(* IEC 61131-3 sources: HappyLearnCodesys/content/softmotion/Robotics_DynamicModel, 17 files *)

(* ---- MatSI_ApplyTwist.st ---- *)
/// Applies a spatial inertia matrix to a twist vector
/// resulting in a generalized momentum or force vector
/// depending on whether the twist represents a velocity
/// or an acceleration.
FUNCTION MatSI_ApplyTwist
VAR_IN_OUT
    /// The resulting generalized momentum or force.
    W : WrenchVec;
END_VAR
VAR_IN_OUT CONSTANT
    /// The spatial inertia matrix.
    G : SMDYN.DynSpatialInertia;
    /// The generalized velocity or acceleration.
    T : TwistVec;
END_VAR

SM3M.SMC_Matrix3_Apply(W.m, G.I, T.w);
SM3M.SMC_V3_Mult(W.f, T.v, G.m);

(* ---- SMC_Frame_ApplyTwist.st ---- *)
/// Applies a coordinate transformation T_ab to a twist vector V_b in se(3).
///       |   mR     0 |
/// V_a = |            | V_b
///       |[vT]*mR   mR|
FUNCTION SMC_Frame_ApplyTwist
VAR_IN_OUT
    /// Twist vector in a frame coordinates
	V_a : TwistVec;
END_VAR
VAR_IN_OUT CONSTANT
    /// Orientation and position of the b frame
    /// in a frame coordinates.
	T_ab : SM3M.SMC_Frame;
    /// Twist vector in b frame coordinates.
	V_b : TwistVec;
END_VAR
VAR
    vTmp : SM3M.SMC_VECTOR3D;
END_VAR

SM3M.SMC_Matrix3_Apply(V_a.w, T_ab.mR, V_b.w);
SM3M.SMC_Matrix3_Apply(V_a.v, T_ab.mR, V_b.v);
SM3M.SMC_V3_Cross(vTmp, T_ab.vT, V_a.w);
SM3M.SMC_V3_Add(V_a.v, V_a.v, vTmp);

(* ---- SMC_Frame_ApplyWrench.st ---- *)
/// Applies a coordinate transformation T_ab to a wrench vector F_a in se(3).
///       |mR^T  mR^T*[vT]^T|
/// F_b = |                 | F_a
///       | 0         mR^T  |
FUNCTION SMC_Frame_ApplyWrench
VAR_IN_OUT
    /// Wrench vector in b frame coordinates.
	F_b : WrenchVec;
END_VAR
VAR_IN_OUT CONSTANT
    /// Orientation and position of the b frame
    /// in a frame coordinates.
	T_ab : SM3M.SMC_Frame;
    /// Wrench vector in a frame coordinates.
	F_a : WrenchVec;
END_VAR
VAR
    mR_ : SM3M.SMC_Matrix3;
    wTmp0 : SM3M.SMC_VECTOR3D;
    wTmp1 : SM3M.SMC_VECTOR3D;
END_VAR

SM3M.SMC_Matrix3_Transpose(mR_, T_ab.mR);
SM3M.SMC_Matrix3_Apply(F_b.m, mR_, F_a.m);
SM3M.SMC_V3_Cross(wTmp0, T_ab.vT, F_a.f);
SM3M.SMC_Matrix3_Apply(wTmp1, mR_, wTmp0);
SM3M.SMC_V3_Sub(F_b.m, F_b.m, wTmp1);

SM3M.SMC_Matrix3_Apply(F_b.f, mR_, F_a.f);

(* ---- SMC_Frame_FromScrewAxisAngle.st ---- *)
/// Calculates an SE(3) frame from a screw axis
/// (a normalized |TwistVec|) and an angle.
FUNCTION SMC_Frame_FromScrewAxisAngle
VAR_IN_OUT
    /// The resulting frame.
    f : SM3M.SMC_Frame;
END_VAR
VAR_IN_OUT CONSTANT
    /// The screw axis.
    A : TwistVec;
END_VAR
VAR_INPUT
    /// The angle.
    theta : LREAL;
END_VAR
VAR
    wv : SM3M.SMC_VECTOR3D;
    w2v : SM3M.SMC_VECTOR3D;
    wt : SM3M.SMC_VECTOR3D;
END_VAR

SM3M.SMC_V3_Cross(wv, A.w, A.v);
SM3M.SMC_V3_Cross(w2v, A.w, wv);

SM3M.SMC_V3_Mult(f.vT, A.v, theta);
SM3M.SMC_V3_MAdd(f.vT, f.vT, wv, (1 - COS(theta)));
SM3M.SMC_V3_MAdd(f.vT, f.vT, w2v, (theta - SIN(theta)));

SM3M.SMC_V3_Mult(wt, A.w, theta);
SM3M.SMC_Matrix3_FromAxisAngle(f.mR, wt);

(* ---- SMC_OpenChainKinematics_SolveForward.st ---- *)
FUNCTION SMC_OpenChainKinematics_SolveForward
VAR_IN_OUT
    fTCP : SM3M.SMC_Frame;
END_VAR
VAR_IN_OUT CONSTANT
    aS : ARRAY[0..SM3M.SMC_MAX_VEC_DIM-1] OF TwistVec;
    vJoints : SM3M.SMC_Vec;
    fTCP_init : SM3M.SMC_Frame;
END_VAR
VAR
    i : UDINT;
    fTmp : SM3M.SMC_Frame;
    afCur : ARRAY[0..1] OF SM3M.SMC_Frame;
END_VAR

i := TO_UDINT(vJoints.n);
afCur[i AND 1] := fTCP_init;
WHILE i > 0 DO
    SMC_Frame_FromScrewAxisAngle(fTmp, aS[i-1], vJoints.a[i-1]);
    SM3M.SMC_Frame_Mult(afCur[(i-1) AND 1], fTmp, afCur[i AND 1]);

    i := i - 1;
END_WHILE

fTCP := afCur[0];

(* ---- Twist_Bracket_Twist.st ---- *)
/// Calculates the generalized cross product
/// between two |TwistVec|s, both representing
/// generalized velocities. The result is a
/// generalized acceleration.
FUNCTION Twist_Bracket_Twist
VAR_IN_OUT
    /// The resulting acceleration.
    V_dst : TwistVec;
END_VAR
VAR_IN_OUT CONSTANT
    /// The first velocity.
    V_lhs : TwistVec;
    /// The second velocity.
    V_rhs : TwistVec;
END_VAR
VAR
    v0 : SM3M.SMC_VECTOR3D;
    v1 : SM3M.SMC_VECTOR3D;
END_VAR

SM3M.SMC_V3_Cross(v0, V_lhs.v, V_rhs.w);
SM3M.SMC_V3_Cross(v1, V_lhs.w, V_rhs.v);
SM3M.SMC_V3_Cross(V_dst.w, V_lhs.w, V_rhs.w);
SM3M.SMC_V3_Add(V_dst.v, v0, v1);

(* ---- Twist_Bracket_Wrench.st ---- *)
/// Calculates the generalized cross product
/// between a |TwistVec|, representing a generalized
/// velocity, and a |WrenchVec|, representing a
/// generalized momentum, resulting in a generalized
/// force.
FUNCTION Twist_Bracket_Wrench
VAR_IN_OUT
    /// The resulting force.
    F_dst : WrenchVec;
END_VAR
VAR_IN_OUT CONSTANT
    /// The velocity.
    V_src : TwistVec;
    /// The momentum.
    F_src : WrenchVec;
END_VAR
VAR
    m0 : SM3M.SMC_VECTOR3D;
    m1 : SM3M.SMC_VECTOR3D;
END_VAR

SM3M.SMC_V3_Cross(m0, F_src.m, V_src.w);
SM3M.SMC_V3_Cross(m1, F_src.f, V_src.v);
SM3M.SMC_V3_Cross(F_dst.f, F_src.f, V_src.w);
SM3M.SMC_V3_Add(F_dst.m, m0, m1);

(* ---- TwistVec_Add.st ---- *)
FUNCTION TwistVec_Add
VAR_IN_OUT
    V_dst : TwistVec;
END_VAR
VAR_IN_OUT CONSTANT
    V_lhs : TwistVec;
    V_rhs : TwistVec;
END_VAR

SM3M.SMC_V3_Add(V_dst.w, V_lhs.w, V_rhs.w);
SM3M.SMC_V3_Add(V_dst.v, V_lhs.v, V_rhs.v);

(* ---- TwistVec_Scale.st ---- *)
FUNCTION TwistVec_Scale
VAR_IN_OUT
    V_dst : TwistVec;
END_VAR
VAR_IN_OUT CONSTANT
    V_src : TwistVec;
END_VAR
VAR_INPUT
    theta : LREAL;
END_VAR

SM3M.SMC_V3_Mult(V_dst.w, V_src.w, theta);
SM3M.SMC_V3_Mult(V_dst.v, V_src.v, theta);

(* ---- Wrench_Dot_Twist.st ---- *)
/// Calculates the dot product between a wrench and a twist.
FUNCTION Wrench_Dot_Twist
VAR_IN_OUT CONSTANT
    F : WrenchVec;
    V : TwistVec;
END_VAR
VAR_OUTPUT
    Wrench_Dot_Twist : LREAL;
END_VAR

Wrench_Dot_Twist := SM3M.SMC_V3_Dot(F.m, V.w) + SM3M.SMC_V3_Dot(F.f, V.v);

(* ---- WrenchVec_Add.st ---- *)
FUNCTION WrenchVec_Add
VAR_IN_OUT
    F_dst : WrenchVec;
END_VAR
VAR_IN_OUT CONSTANT
    F_lhs : WrenchVec;
    F_rhs : WrenchVec;
END_VAR

SM3M.SMC_V3_Add(F_dst.m, F_lhs.m, F_rhs.m);
SM3M.SMC_V3_Add(F_dst.f, F_lhs.f, F_rhs.f);

(* ---- WrenchVec_Sub.st ---- *)
FUNCTION WrenchVec_Sub
VAR_IN_OUT
    V_dst : WrenchVec;
END_VAR
VAR_IN_OUT CONSTANT
    V_lhs : WrenchVec;
    V_rhs : WrenchVec;
END_VAR

SM3M.SMC_V3_Sub(V_dst.m, V_lhs.m, V_rhs.m);
SM3M.SMC_V3_Sub(V_dst.f, V_lhs.f, V_rhs.f);

(* ---- DynModel_Scara2_Z.st ---- *)
(*
    檔案用途：
      定義一具 3 自由度 Scara+Z 機構的動力學模型，包含各連桿的幾何尺寸、
      質量、慣性矩與螺旋軸（screw axes），並實作 SMDYN.ISMDynamics 介面，
      供 SoftMotion 的動力學模組計算關節扭矩與負載效應。
    教學重點：
      - 觀察 m_aM（各連桿質心座標）、m_aG（空間慣性）、m_aS（螺旋軸）三組資料的物理意義。
      - 理解 DOF 與臂長／質量等常數，如何對應到實際 Scara 幾何結構。
      - 作為自訂機構動力學定義的範例，供其他機構參考套用。
*)
FUNCTION_BLOCK DynModel_Scara2_Z IMPLEMENTS SMDYN.ISMDynamics
VAR CONSTANT
	/// Degrees of freedom.
	DOF : DINT := 3;
	/// All length values in [m]
	armOneLength : LREAL := 0.4;
	armTwoLength : LREAL := 0.3;
	baseHeight : LREAL := 0.6;
	armOneHeight : LREAL := 0.06;
	armTwoHeight : LREAL := 0.06;
	zAxisLength : LREAL := 0.3;
	zAxisOffset : LREAL := -0.05;
	/// All mass values in [kg]
	armOneMass : LREAL := 3;
	armTwoMass : LREAL := 4;
	zAxisMass : LREAL := 1;

	/// The home position of all link frames. |aM[i]| contains
    /// the frame of the ith link expressed in the coordinates of the
    /// (i-1)th link frame.
    /// All frames are expected to be situated at the link's center
    /// of mass.
    m_aM : ARRAY[0..SMRB.MAX_VEC_DIM] OF SM3M.SMC_Frame := [
        /// All values of vT in [m]
        ///
        /// The center of mass of arm 1 expressed in the base coordinate system 0:
        (mR:= (
            aElems:= [
                1, 0, 0,
                0, -1, 0,
                0, 0, -1]),
         vT:= (dX:= armOneLength / 2.0, dY:= 0, dZ:= baseHeight + armOneHeight / 2.0)),
        /// The center of mass of arm 2 expressed in the coordinate system of arm 1:
        (mR:= (
            aElems:= [
                1, 0, 0,
                0, 1, 0,
                0, 0, 1]),
         vT:= (dX:= armOneLength / 2.0 + armTwoLength / 2.0, dY:= 0, dZ:= armOneHeight / 2.0 + armTwoHeight / 2.0)),
        /// The center of mass of the z-axis expressed in the coordinate system of arm 2:
        (mR:= (
            aElems:= [
                1, 0, 0,
                0, 1, 0,
                0, 0, 1]),
         vT:= (dX:= armTwoLength / 2.0, dY:= 0, dZ:= zAxisLength / 2.0 - armTwoHeight / 2.0 + zAxisOffset)),
        /// One additional array entry, to handle an arbitrary load at the TCP, expressed
		/// in the coordinate system of the z-axis.
        (mR:= (
            aElems:= [
                1, 0, 0,
                0, 1, 0,
                0, 0, 1]),
         vT:= (dX:= 0, dY:= 0, dZ:= - zAxisLength / 2.0))];

	/// The spatial inertia matrices of all links, expressed in the
    /// respectives link's frame.
    m_aG : ARRAY[0..SMRB.MAX_VEC_DIM-1] OF SMDYN.DynSpatialInertia := [
        /// All inertia values in [kg m²]
        /// and all mass values in [kg]
        /// Arm 1
        (I:= (
            aElems:= [
                0, 0, 0,
                0, 1/12.0 * armOneMass * armOneLength * armOneLength, 0,
                0, 0, 1/12.0 * armOneMass * armOneLength * armOneLength]),
         m:= armOneMass),
        /// Arm 2
        (I:= (
            aElems:= [
                0, 0, 0,
                0, 1/12.0 * armTwoMass * armTwoLength * armTwoLength, 0,
                0, 0, 1/12.0 * armTwoMass * armTwoLength * armTwoLength]),
         m:= armTwoMass),
        /// z-axis
        (I:= (
            aElems:= [
                1/12.0 * zAxisMass * zAxisLength * zAxisLength, 0, 0,
                0, 1/12.0 * zAxisMass * zAxisLength * zAxisLength, 0,
                0, 0, 0]),
         m:= zAxisMass)];

	/// The screw axes of all joints, expressed in the base frame.
    m_aS : ARRAY[0..SMRB.MAX_VEC_DIM-1] OF TwistVec := [
		/// Angular velocities in [rad/s] and linear velocities in [m/s].
        /// Screw axis of arm 1
        (w:= (dX:= 0, dY:= 0, dZ:= 1),
         v:= (dX:= 0, dY:= 0, dZ:= 0)),
        /// Screw axis of arm 2
        (w:= (dX:= 0, dY:= 0, dZ:= 1),
         v:= (dX:= 0, dY:= -armOneLength, dZ:= 0)),
        /// Screw axis of the z-axis
        (w:= (dX:= 0, dY:= 0, dZ:= 0),
         v:= (dX:= 0, dY:= 0, dZ:= 1))];
END_VAR
VAR
    /// The home position of all link frames. |m_aM_inv[i]| contains
    /// the frame of the (i-1) link expressed in the coordinates of the
    /// ith link frame.
    /// All frames are expected to be situated at the link's center
    /// of mass.
    m_aM_inv : ARRAY[0..SM3M.SMC_MAX_VEC_DIM] OF SM3M.SMC_Frame;
    /// The screw axes of all joints, expressed in the link's frame.
    m_aA : ARRAY[0..SM3M.SMC_MAX_VEC_DIM-1] OF TwistVec;
END_VAR

(* ---- SetAxisLimits.st ---- *)
FUNCTION_BLOCK SetAxisLimits
VAR_IN_OUT
	AxisGroup : AXIS_GROUP_REF_SM3;
END_VAR
VAR_INPUT
	Execute : BOOL;
	AxisLimits : ARRAY[0..SMC_RCNST.MAX_AXES-1] OF AxisLimits;
END_VAR
VAR_OUTPUT
	Done : BOOL;
	Error : BOOL;
	ErrorID : SMC_ERROR;
END_VAR
VAR
	state : INT := IDLE_STATE;

	groupDisable : MC_GroupDisable;
	groupEnable : MC_GroupEnable;
	groupStatus : MC_GroupReadStatus;
	groupReadConfig : MC_GroupReadConfiguration;
	changeDynamicLimits : SMC_ChangeDynamicLimits;

	currentAxis : IDENT_IN_GROUP_REF_SM3;
	oldExecute : BOOL;
END_VAR
VAR CONSTANT
	IDLE_STATE : INT := 0;
	CHECK_STATE : INT := 10;
	DISABLE_STATE : INT := 20;
	READ_CONFIG_STATE : INT := 30;
	CHANGE_DYNAMIC_LIMIT_STATE : INT := 40;
	PREPARE_NEXT_AXIS_STATE : INT := 50;
	ENABLE_STATE : INT := 60;
	DONE_STATE : INT := 100;
	ERROR_STATE : INT := 1000;
END_VAR

IF Execute AND_THEN NOT oldExecute THEN
	state := CHECK_STATE;
	currentAxis := 0;
	ErrorID := SMC_NO_ERROR;
ELSIF NOT Execute
	AND_THEN (state = DONE_STATE OR_ELSE state = ERROR_STATE)
THEN
	state := IDLE_STATE;
	ErrorID := SMC_NO_ERROR;
END_IF

CASE state OF
	CHECK_STATE:
		IF groupStatus.Valid AND_THEN groupStatus.GroupStandby THEN
			state := DISABLE_STATE;
		ELSIF groupStatus.Valid THEN
			state := READ_CONFIG_STATE;
		END_IF

	DISABLE_STATE:
		groupDisable.Execute := TRUE;

		IF groupDisable.Done THEN
			groupDisable.Execute := FALSE;
			state := READ_CONFIG_STATE;
		ELSIF groupDisable.Error THEN
			groupDisable.Execute := FALSE;
			state := ERROR_STATE;
			ErrorID := groupDisable.ErrorID;
		END_IF

	READ_CONFIG_STATE:
		groupReadConfig(
			AxisGroup:= AxisGroup,
			Enable:= TRUE,
			IdentInGroup:= currentAxis);

		IF groupReadConfig.Valid THEN
			state := CHANGE_DYNAMIC_LIMIT_STATE;
		ELSIF groupReadConfig.Error THEN
			state := ERROR_STATE;
			ErrorID := groupReadConfig.ErrorID;
		END_IF

	CHANGE_DYNAMIC_LIMIT_STATE:
		changeDynamicLimits(
			Axis:= groupReadConfig.pAxis^,
			bExecute:= TRUE,
			fMaxVelocity:= AxisLimits[currentAxis].maxVelocity,
			fMaxAcceleration:= AxisLimits[currentAxis].maxAcceleration,
			fMaxDeceleration:= AxisLimits[currentAxis].maxDeceleration,
			fMaxJerk:= AxisLimits[currentAxis].maxJerk,
			fMaxTorque:= AxisLimits[currentAxis].maxTorque);

		IF changeDynamicLimits.bDone THEN
			changeDynamicLimits(Axis:= groupReadConfig.pAxis^, bExecute:= FALSE);
			state := PREPARE_NEXT_AXIS_STATE;
		ELSIF changeDynamicLimits.bError THEN
			state := ERROR_STATE;
			ErrorID := changeDynamicLimits.ErrorID;
			changeDynamicLimits(Axis:= groupReadConfig.pAxis^, bExecute:= FALSE);
		END_IF

	PREPARE_NEXT_AXIS_STATE:
		currentAxis := currentAxis + 1;

		IF currentAxis < groupReadConfig.NumAxes THEN
			state := READ_CONFIG_STATE;
		ELSE
			state := ENABLE_STATE;
		END_IF

	ENABLE_STATE:
		groupEnable.Execute := TRUE;

		IF groupEnable.Done THEN
			groupEnable.Execute := FALSE;
			state := DONE_STATE;
		ELSIF groupEnable.Error THEN
			groupEnable.Execute := FALSE;
			state := ERROR_STATE;
			ErrorID := groupEnable.ErrorID;
		END_IF
END_CASE

groupDisable(AxisGroup:= AxisGroup);
groupEnable(AxisGroup:= AxisGroup);
groupStatus(AxisGroup:= AxisGroup, Enable:= TRUE);

Done := state = DONE_STATE;
Error := state = ERROR_STATE;

oldExecute := Execute;

(* ---- Test_DynModel_Scara2_Z.st ---- *)
FUNCTION_BLOCK Test_DynModel_Scara2_Z
VAR
	m_dynModel : DynModel_Scara2_Z;
END_VAR
VAR CONSTANT
	/// Frame of the initial robot position.
	ZERO_TCP_FRAME : SM3M.SMC_Frame := (
        mR:= (
            aElems:= [
                1, 0, 0,
                0, 1, 0,
                0, 0, 1]),
        vT:= (
			dX:= m_dynModel.armOneLength + m_dynModel.armTwoLength,
			dY:= 0,
			dZ:= - m_dynModel.baseHeight - m_dynModel.armOneHeight - m_dynModel.zAxisOffset));
END_VAR

(* ---- DynModel_Tests.st ---- *)
(*
    檔案用途：
      透過 Test_DynModel_Scara2_Z 功能塊，對 Scara 動力學模型做單元測試，
      包含檢查螺旋軸定義（CheckScrewAxis）與靜止扭矩計算（CheckStandstillTorque）。
    教學重點：
      - 示範如何以簡單狀態機包裝一組動力學測試，將結果輸出為 successful / error。
      - 幫助使用者在將模型套用到 PLC_PRG 前，先驗證模型本身是否合理。
*)
PROGRAM DynModel_Tests
VAR_OUTPUT
	successful: BOOL;
	error : BOOL;
END_VAR
VAR
	state : INT;
	tester : Test_DynModel_Scara2_Z;
END_VAR

CASE state OF
	0:
		IF tester.CheckScrewAxis() THEN
			state := state + 10;
		ELSE
			state := state + 1000;
		END_IF

	10:
		IF tester.CheckStandstillTorque() THEN
			state := state + 10;
		ELSE
			state := state + 1000;
		END_IF

	20:
		state := 100;
END_CASE

successful := state = 100;
error := state >= 1000;

(* ---- PLC_PRG.st ---- *)
(*
    檔案用途：
      示範如何在 SoftMotion 中使用自訂的動力學模型（DynModel_Scara2_Z），
      針對相同的關節移動，比較「無扭矩限制」、「有限扭矩」、「加掛負載」三種情境下
      軸的速度／加速度／扭矩行為差異。
    教學重點：
      - 看懂 TorqueLimitationDemoStates 狀態機如何分段執行三種測試運動。
      - 理解 SMC_GroupSetDynamics、SMC_GroupSetLoad、SetAxisLimits 搭配使用的方式。
      - 練習從 TEST_MOVEMENT_* 的設定與 Trace 變數中，觀察動力學模型對實際運動的影響。
*)
PROGRAM PLC_PRG
VAR
	state : TorqueLimitationDemoStates;

	currentTestMovement : UINT := 0;
	start : SMC_POS_REF;
	destination : SMC_POS_REF;

	groupPower : SMC_GroupPower;
	setDynamics : SMC_GroupSetDynamics;
	dynModel : DynModel_Scara2_Z;
	moveDirectAbs : MC_MoveDirectAbsolute := (CoordSystem:= SMC_COORD_SYSTEM.ACS);
	setLoad : SMC_GroupSetLoad := (ExecutionMode:= MC_EXECUTION_MODE.Immediately);
	setPosition : MC_GroupSetPosition;
	setAxisLimits : SetAxisLimits;
END_VAR
VAR CONSTANT
	/// Count of different test movements.
	TEST_MOVEMENT_COUNT : UINT := 2;

	/// Load mass in [kg]
	LOAD_MASS : LREAL := 3;
	/// Load length in [m]
	LOAD_LENGTH : LREAL := 0.2;
	/// Load calculated for a thin rod mounted directly
	/// to the z-axis in [kg m²]
	LOAD : SMC_DynLoad :=
		(
			Mass:= LOAD_MASS,
			PrincipalMoments:=
				[
					/// Ix
					0,
					/// Iy
					1/12.0 * LOAD_MASS * LOAD_LENGTH * LOAD_LENGTH,
					/// Iz
					1/12.0 * LOAD_MASS * LOAD_LENGTH * LOAD_LENGTH
				]
		);
	ZERO_LOAD : SMC_DynLoad :=
		(
			Mass:= 0,
			PrincipalMoments:= [0, 0, 0],
			PrincipalAxes:= (X:= 0, Y:= 0, Z:= 0, A:= 0, B:= 0, C:= 0)
		);

	/// Test movement positions in ACS (a0 and a1 in [°] and a2 in [m]).
	TEST_MOVEMENT_ONE_START : SMC_POS_REF := (a:= (a0:= 0, a1:= 0, a2:= 0));
	TEST_MOVEMENT_ONE_DESTINATION : SMC_POS_REF := (a:= (a0:= 90, a1:= 0, a2:= 0.02));
	TEST_MOVEMENT_TWO_START : SMC_POS_REF := (a:= (a0:= 0, a1:= -120, a2:= 0));
	TEST_MOVEMENT_TWO_DESTINATION : SMC_POS_REF := (a:= (a0:= 90, a1:= -120, a2:= 0.02));

	DEFAULT_REVOLUTE_AXIS_LIMITS : AxisLimits :=
		(
			maxVelocity:= 30,	/// [°/s]
			maxAcceleration:= 400,	/// [°/s²]
			maxDeceleration:= 400,	/// [°/s²]
			maxJerk:= 1E5,	/// [°/s³]
			maxTorque:= FPU.GetLRealSpecialVal(FPU.ESpecial_FP_Value.PosInf)	/// [Nm]
		);

	DEFAULT_PRISMATIC_AXIS_LIMITS : AxisLimits :=
		(
			maxVelocity:= 0.03,	/// [m/s]
			maxAcceleration:= 0.4,	/// [m/s²]
			maxDeceleration:= 0.4,	/// [m/s²]
			maxJerk:= 10,	/// [m/s³]
			maxTorque:= FPU.GetLRealSpecialVal(FPU.ESpecial_FP_Value.PosInf)	/// [N]
		);
END_VAR

CASE state OF
	PowerAxisGroup:
		groupPower.bDriveStart := TRUE;
		groupPower.bRegulatorOn := TRUE;
		groupPower.Enable := TRUE;

		IF groupPower.Status THEN
			state := InitializeDynamicModel;
		END_IF

	InitializeDynamicModel:
		dynModel.Init();

		setDynamics.Dynamics := dynModel;
		/// Gravitational acceleration in [m/s²]
		setDynamics.GravitationalAcceleration.dZ := 9.81;
		setDynamics.Execute := TRUE;

		IF setDynamics.Done THEN
			state := InitializeTestMovement;
		END_IF

	InitializeTestMovement:
		CASE currentTestMovement OF
			0:
				start := TEST_MOVEMENT_ONE_START;
				destination := TEST_MOVEMENT_ONE_DESTINATION;
			1:
				start := TEST_MOVEMENT_TWO_START;
				destination := TEST_MOVEMENT_TWO_DESTINATION;
		END_CASE

		setLoad.Load := ZERO_LOAD;
		setLoad.Execute := TRUE;

		IF setLoad.Done THEN
			setLoad.Execute := FALSE;
			state := InitializeUnlimitedTorqueMovement;
		END_IF

	InitializeUnlimitedTorqueMovement:
		setAxisLimits.AxisLimits[0] := DEFAULT_REVOLUTE_AXIS_LIMITS;
		setAxisLimits.AxisLimits[1] := DEFAULT_REVOLUTE_AXIS_LIMITS;
		setAxisLimits.AxisLimits[2] := DEFAULT_PRISMATIC_AXIS_LIMITS;

		setAxisLimits.Execute := TRUE;

		IF setAxisLimits.Done AND_THEN ResetRobotPosition() THEN
			setAxisLimits.Execute := FALSE;
			state := ExecuteUnlimitedTorqueMovement;
		END_IF

	ExecuteUnlimitedTorqueMovement:
		moveDirectAbs.Position := destination;
		moveDirectAbs.Execute := TRUE;

		IF moveDirectAbs.Done THEN
			moveDirectAbs.Execute := FALSE;
			state := InitializeLimitedTorqueMovement;
		END_IF

	InitializeLimitedTorqueMovement:
		/// Torque limit for axis 2 in [Nm]
		setAxisLimits.AxisLimits[1].maxTorque := 2;
		setAxisLimits.Execute := TRUE;

		IF setAxisLimits.Done AND_THEN ResetRobotPosition() THEN
			setAxisLimits.Execute := FALSE;
			state := ExecuteLimitedTorqueMovement;
		END_IF

	ExecuteLimitedTorqueMovement:
		moveDirectAbs.Position := destination;
		moveDirectAbs.Execute := TRUE;

		IF moveDirectAbs.Done THEN
			moveDirectAbs.Execute := FALSE;
			state := InitializeMovementWithLoad;
		END_IF

	InitializeMovementWithLoad:
		setLoad.Load := LOAD;
		setLoad.Execute := TRUE;

		IF setLoad.Done AND_THEN ResetRobotPosition() THEN
			setLoad.Execute := FALSE;
			state := ExecuteMovementWithLoad;
		END_IF

	ExecuteMovementWithLoad:
		moveDirectAbs.Position := destination;
		moveDirectAbs.Execute := TRUE;

		IF moveDirectAbs.Done THEN
			moveDirectAbs.Execute := FALSE;
			state := FinalizeTestMovement;
		END_IF

	FinalizeTestMovement:
		currentTestMovement := currentTestMovement + 1;

		IF currentTestMovement < TEST_MOVEMENT_COUNT THEN
			state := InitializeTestMovement;
		ELSE
			state := DemoFinished;
		END_IF
END_CASE

groupPower(AxisGroup:= AxisGroup);
setDynamics(AxisGroup:= AxisGroup);
moveDirectAbs(AxisGroup:= AxisGroup);
setLoad(AxisGroup:= AxisGroup);
setPosition(AxisGroup:= AxisGroup);
setAxisLimits(AxisGroup:= AxisGroup);
